FUNCTION_BLOCK ReadCoordinates EXTENDS TcoCore.TcoTask
VAR_IN_OUT
    InfoData       : InfoData_32EB74EA;
    StatusOfSystem : Status_of_System;
    ResultValue    : DINT;
END_VAR
VAR_INPUT
    ActionDesc : STRING(25);
END_VAR
VAR
    _fb_coe_read_ext         : Tc2_EtherCAT.FB_EcCoESdoReadEx;
    _timeout                 : TIME := Tc2_System.DEFAULT_ADS_TIMEOUT;
    _state                   : INT  := 10;
    _data                    : ARRAY[1..31] OF DINT;
    _errorId                 : UDINT;
    _rawCoordinates          : Coordinates;
    _coeIndex                : UINT;
    _distanceFromHeight      : LREAL;
    _fieldOfView             : FieldOfView;
    _coordinatesInMillimeter : Coordinates;
END_VAR
VAR CONSTANT
    SIZE_OF_TWO_BYTES : UINT := 16;
    ResolutionX       : UINT := 1280;
    ResolutionY       : UINT := 960;

END_VAR


IF (THIS^.Execute()) THEN
    //ERror Case

    THIS^.ThrowWhen(StatusOfSystem.Error_Status);

    CASE _state OF
        10:
            _fb_coe_read_ext
            (
                sNetId            := Tc2_System.F_CreateAmsNetId(infodata.AdsAddr.netId)
                , nSlaveAddr      := InfoData.AdsAddr.port
                , nSubIndex       := 16#0
                , nIndex          := _coeIndex
                , pDstBuf         := ADR(_data)
                , cbBufLen        := SIZEOF(_data) + 2
                , tTimeout        := _timeout
                , bCompleteAccess := TRUE
            );

            _state := 20;
        20:
            _fb_coe_read_ext(bExecute := TRUE);
            _state := 30;
        30:
            _fb_coe_read_ext();

            IF _fb_coe_read_ext.bBusy THEN
                RETURN;
            END_IF

            IF _fb_coe_read_ext.bError THEN
                _State := 99; // Error case
                RETURN;
            END_IF

            _rawCoordinates.xValue        := SHR(_data[017], SIZE_OF_TWO_BYTES);
            _rawCoordinates.yValue        := SHR(_data[018], SIZE_OF_TWO_BYTES);
            _rawCoordinates.variableValue := SHR(_data[019], SIZE_OF_TWO_BYTES);

            _state := 40;
        40:
            DistanceFromHeight
            (
                Resolution    := ResolutionY
                , Pixel       := _rawCoordinates.variableValue
                , Height      := THIS^.ResultValue 
                , FieldOfView => _fieldOfView
                , Distance    => _distanceFromHeight
            );

            _state := 50;
        50:

            THIS^.DoneWhen(TRUE);
        99:
            THIS^.ThrowWhen(TRUE);

    END_CASE
END_IF

METHOD PROTECTED CalcCoefficientFromResolutionAndPixel : LREAL
VAR_INPUT
    Resolution : LREAL;
    Pixel      : LREAL;
END_VAR

IF Pixel = 0 THEN
    THIS^.Messenger.Error('Was ist los mit dir, teile nicht durch 0!');
    CalcCoefficientFromResolutionAndPixel := 0;
    RETURN;
END_IF

CalcCoefficientFromResolutionAndPixel := (Resolution / Pixel) * 10;
END_METHOD

METHOD PRIVATE CalcFieldOfViewWithCoefficientAndObjectMeasurement : LREAL
VAR_INPUT
    Coefficient : LREAL;
    Height      : DINT;
END_VAR
CalcFieldOfViewWithCoefficientAndObjectMeasurement := (Coefficient * DWORD_TO_LREAL(Height)) / 100;
END_METHOD

PROPERTY CoordinatesInMillimeter: REFERENCE TO Coordinates
GET
CoordinatesInMillimeter Ref= _coordinatesInMillimeter;
END_GET
END_PROPERTY

METHOD PRIVATE DistanceFromHeight
VAR_OUTPUT
    FieldOfView : FieldOfView;
    Distance    : LREAL;
END_VAR
VAR_INPUT
    Resolution : LREAL;
    Pixel      : LREAL;
    Height     : DINT;
END_VAR
VAR_INST
    //lineare Regression
    offset      : LREAL := -5.57888;
    gain        : LREAL := 3.387877;
    Coefficient : LREAL;
END_VAR
//in mm     Breite
//50		16,4		
//100		31,2		
//200		60,7		
//300		90,2		
//400		119,7		
//500		149,2		
//600		178,7		
//700		208,3		
//800		237,8		
//900		267,3		
//1000		296,8	
//1250		370,6	
//1500		444,4	
//1750		518,2	
//2000		592
// Resolution / Pixel = Coefficient
//Coefficient * Length = FieldOfView
// With FOV calculate the Distance of the Object to the Sensor
//Distance = (FOV-b)/m
if Pixel = 0 then
    ;
ELSE
    Coefficient := CalcCoefficientFromResolutionAndPixel(Resolution := Resolution, Pixel := Pixel);

    FieldOfView.yValue := CalcFieldOfViewWithCoefficientAndObjectMeasurement
    (
        Coefficient := Coefficient
        , Height    := Height
    );

    Distance := (FieldOfView.yValue * gain) + offset;
END_IF
END_METHOD

PROPERTY DistanceFromObject : LREAL
GET
DistanceFromObject := _distanceFromHeight;
END_GET
END_PROPERTY

{attribute 'monitoring' := 'call'}
PROPERTY ErrorId : UINT
GET
ErrorId := udint_to_uint(_errorId);
END_GET
END_PROPERTY

METHOD PUBLIC FB_init : BOOL
VAR_INPUT
    bInitRetains : BOOL; // if TRUE, the retain variables are initialized (warm start / cold start)
    bInCopyCode  : BOOL; // if TRUE, the instance afterwards gets moved into the copy code (online change)
    ParentObject : ITcoObject;
    CoeIndex     : UINT;
END_VAR
// This is not clear to me... I from time to time the consumer code does not see 'FB_init' of 'TcoObject', that's why overridden here with super call...
{warning disable C0316}
SUPER^.FB_init(bInitRetains, bInCopyCode, ParentObject);

_coeIndex         := CoeIndex;
END_METHOD

PROPERTY FieldOfView : REFERENCE TO FieldOfView
GET
FieldOfView REF= _fieldOfView;
END_GET
END_PROPERTY

(*~
    <docu>
        <summary>
            Executes when task reaches the ```Done``` state .
        </summary>
    </docu>
~*)
METHOD PROTECTED OnDone
{warning disable C0371}
_fb_coe_read_ext(bExecute := False);
END_METHOD

(*~
    <docu>
        <summary>
            Executes when task reaches the ```Error``` state.
            <para>
                Do not confuse with <see cref="PlcDocu.TcoCore.TcoTask.WhileError()"/>, that is called cyclically until '''Error''' state is left.
            </para>
        </summary>
    </docu>
~*)
METHOD PROTECTED OnError
{warning disable C0371}
_fb_coe_read_ext(nErrId => _errorId);
END_METHOD

(*~
	<docu>
		<summary>
			Executes ones when the task starts (at the moment of transition from the ```Requested``` state into the ```Busy``` state).
		</summary>			
	</docu>	
~*)
METHOD PROTECTED OnStart
{warning disable C0371}
_fb_coe_read_ext(bExecute := FALSE);
_state := 10;
END_METHOD

PROPERTY RawCoordinates : REFERENCE TO Coordinates
GET
RawCoordinates REF= _rawCoordinates;
END_GET
END_PROPERTY

(*~
    <docu>
        <summary>
            Restores this instance to the Ready state. Can be called explicitly or from within one of the restore mechanisms.
            <para>
                See also <see cref="PlcDocu.TcoCore.TcoTask.AutoRestorable()"/>
            </para>
        </summary>
    </docu>
~*)
METHOD Restore : ITcoRestorable
{warning disable C0371}
_fb_coe_read_ext(bExecute := FALSE);
END_METHOD

END_FUNCTION_BLOCK

(* stored: Version 1.1.0.1, ProductVersion 3.1.4024.12
   POU ReadCoordinates: Id {d83738c9-7cff-0c4f-1efe-086a22bcf87d}, SpecialFunc None
   Folder Calculation: Id {96ef91d7-efbb-03c2-2ac3-5a4d4671c693}
   Folder Data: Id {e0b6aee7-66f0-056b-2996-f7cbb14397ea}
   Folder Status: Id {4eca030c-7062-0dd6-349a-bd1a1711aa69}
   Folder TcOpen: Id {40647fab-a281-09f1-3fc9-9c13dbcf1fe1}
   Method CalcCoefficientFromResolutionAndPixel: Id {01de50cb-748a-09b1-3db4-d3ed621575b9}
   Method CalcFieldOfViewWithCoefficientAndObjectMeasurement: Id {69ecf6b6-e253-0fc5-1524-20b5423151cb}
   Property CoordinatesInMillimeter: Id {458c2b93-c4ce-0390-1b53-59fb42433448}
   Get Get: Id {03d8fcde-5f0a-08ee-0862-eda0d7135881}
   Method DistanceFromHeight: Id {dfccd550-8deb-0b1c-0956-40e0bd8ccc01}
   Property DistanceFromObject: Id {aee7e2bd-6ce6-0f90-1195-594df40573f1}
   Get Get: Id {ffc61c06-81f9-04af-2b60-94384cabd68d}
   Property ErrorId: Id {b9119104-ded0-043b-25ee-e9d4629d40a2}
   Get Get: Id {4c55bcce-efca-073a-2133-3e1f9bcc567c}
   Method FB_init: Id {7b6222fc-0c53-0d03-2421-ec4772f70149}
   Property FieldOfView: Id {c2ac5c77-7f0d-00fd-2123-c8e4da7e3178}
   Get Get: Id {be6ceab3-e4f2-0008-1254-217b6672f55b}
   Method OnDone: Id {0ddc4aae-67b7-0e6e-3397-57c4de466ff6}
   Method OnError: Id {baa208b5-517a-0c09-01dc-7068ac8aacaf}
   Method OnStart: Id {104cd4e9-c1b3-0519-18a9-370aec7e8ef2}
   Property RawCoordinates: Id {51be719b-6e54-0146-1c40-0919ea6b3cd5}
   Get Get: Id {c2b1c109-4dae-097e-03a4-318982f4b21e}
   Method Restore: Id {8b9a32c2-68d9-0c41-0b6d-edb4868295bd} *)
